// SIMATIC STEP 7 (V5.x) project verinDuConvoyeurFleche
// CPU: CPU313 C-2 DP(1)
// station: P_ADR_BUS
// station: Hardware
// station: SIMATIC 300 Station
// program: S7 Program(1)

SYMBOL_TABLE
"Marche"	I 0.0	BOOL	// Lancer le système
"Arret"	I 0.1	BOOL	// Arreter le système
"Levée"	I 0.2	BOOL	// Sortir le vérin et lever le convoyeur Flèche
"Descente"	I 0.3	BOOL	// Rentrer le vérin et descendre le convoyeur Flèche
"Vérin En Début"	I 0.4	BOOL
"Vérin En Fin"	I 0.5	BOOL
"Situation Marche"	M 0.0	BOOL	// Le système est activé
"Situation Arret"	M 0.1	BOOL	// Le système est desactivé
"Demande Arret"	M 0.2	BOOL	// Une demande d'arret est faite
"Cycle Execution"	OB 1	OB 1
"Lampe Fonctionnement"	Q 0.0	BOOL	// Visualisation de l'état du système
"Extension Vérin"	Q 0.1	BOOL	// Extension du vérin
"Rétraction Vérin"	Q 0.2	BOOL	// Rétraction du vérin
END_SYMBOL_TABLE

FUNCTION_BLOCK FB 1
TITLE = Situation Système
//Ce programme a comme rôle le control de l'état marche, l'état arret et la 
//demande d'arret du système.
VERSION : 0.1
BEGIN
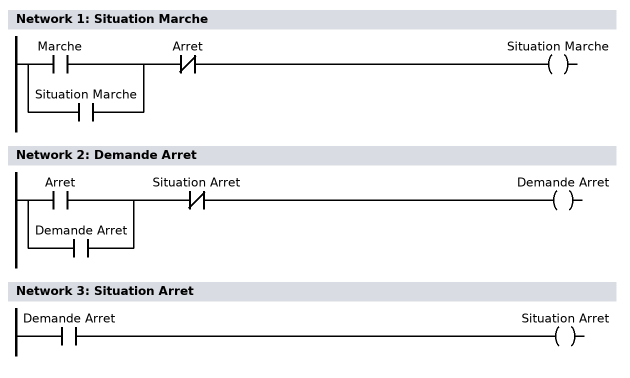
NETWORK
TITLE = Situation Marche
      A(;
      O     "Marche";
      O     "Situation Marche";
      );
      AN    "Arret";
      =     "Situation Marche";
NETWORK
TITLE = Demande Arret
      A(;
      O     "Arret";
      O     "Demande Arret";
      );
      AN    "Situation Arret";
      =     "Demande Arret";
NETWORK
TITLE = Situation Arret
      A     "Demande Arret";
      =     "Situation Arret";
END_FUNCTION_BLOCK

FUNCTION_BLOCK FB 2
TITLE = Extension Vérin
//Le but de ce programme est de controller l'extension du vérin du convoyeur 
//Flèche.
VERSION : 0.1
BEGIN
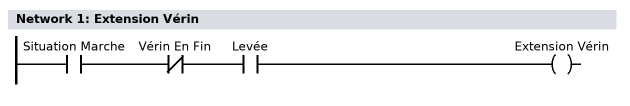
NETWORK
TITLE = Extension Vérin
      A     "Situation Marche";
      AN    "Vérin En Fin";
      A     "Levée";
      =     "Extension Vérin";
END_FUNCTION_BLOCK

FUNCTION_BLOCK FB 3
TITLE = Rétraction Vérin
//Le but de ce programme est de controller la rétraction du vérin du convoyeur 
//Flèche.
VERSION : 0.1
BEGIN
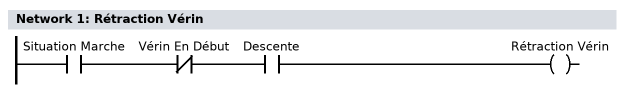
NETWORK
TITLE = Rétraction Vérin
      A     "Situation Marche";
      AN    "Vérin En Début";
      A     "Descente";
      =     "Rétraction Vérin";
END_FUNCTION_BLOCK

FUNCTION_BLOCK FB 4
TITLE = Fonctionnement Visualisation
//Ce programme donne une visualisation sur le fonctionnement des différents 
//programmes.
VERSION : 0.1
BEGIN
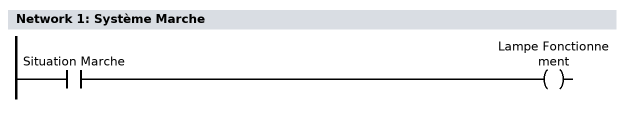
NETWORK
TITLE = Système Marche
      A     "Situation Marche";
      =     "Lampe Fonctionnement";
END_FUNCTION_BLOCK

DATA_BLOCK DB 1
VERSION : 0.0
FB 1
BEGIN
END_DATA_BLOCK

DATA_BLOCK DB 2
VERSION : 0.0
FB 2
BEGIN
END_DATA_BLOCK

DATA_BLOCK DB 3
VERSION : 0.0
FB 3
BEGIN
END_DATA_BLOCK

DATA_BLOCK DB 4
VERSION : 0.0
FB 4
BEGIN
END_DATA_BLOCK

ORGANIZATION_BLOCK "Cycle Execution"	// OB 1
TITLE = "Main Program Sweep (Cycle)"
//Cela est le programme principal qui va être en éxecution infinie.
VERSION : 0.1
VAR_TEMP
  OB1_EV_CLASS : BYTE ;	//Bits 0-3 = 1 (Coming event), Bits 4-7 = 1 (Event class 1)
  OB1_SCAN_1 : BYTE ;	//1 (Cold restart scan 1 of OB 1), 3 (Scan 2-n of OB 1)
  OB1_PRIORITY : BYTE ;	//Priority of OB Execution
  OB1_OB_NUMBR : BYTE ;	//1 (Organization block 1, OB1)
  OB1_RESERVED_1 : BYTE ;	//Reserved for system
  OB1_RESERVED_2 : BYTE ;	//Reserved for system
  OB1_PREV_CYCLE : INT ;	//Cycle time of previous OB1 scan (milliseconds)
  OB1_MIN_CYCLE : INT ;	//Minimum cycle time of OB1 (milliseconds)
  OB1_MAX_CYCLE : INT ;	//Maximum cycle time of OB1 (milliseconds)
  OB1_DATE_TIME : DATE_AND_TIME ;	//Date and time OB1 started
END_VAR
BEGIN
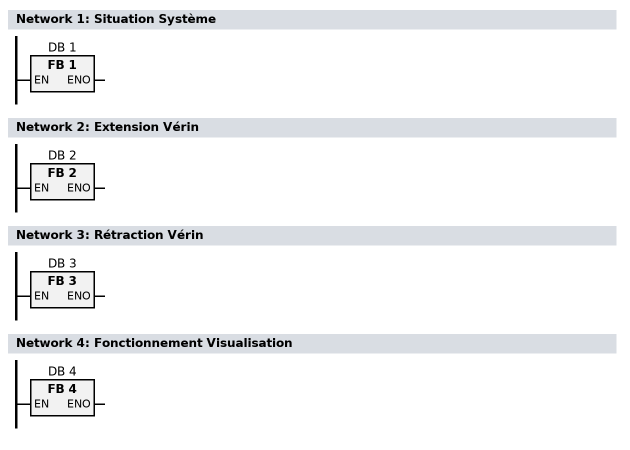
NETWORK
TITLE = Situation Système
      CALL  FB 1 , DB 1;
      NOP   0;
NETWORK
TITLE = Extension Vérin
      CALL  FB 2 , DB 2;
      NOP   0;
NETWORK
TITLE = Rétraction Vérin
      CALL  FB 3 , DB 3;
      NOP   0;
NETWORK
TITLE = Fonctionnement Visualisation
      CALL  FB 4 , DB 4;
      NOP   0;
END_ORGANIZATION_BLOCK
